(* IEC 61131-3 sources: rusty/examples, 13 files *)

(* ---- pointer.st ---- *)
TYPE MyStruct: STRUCT  x: DINT; y: DINT; END_STRUCT END_TYPE

FUNCTION main : DINT
	main := foo();
END_FUNCTION

FUNCTION foo : DINT
VAR
				x : DINT;
				s : MyStruct;
				u,y : REF_TO DINT;
				z : REF_TO REF_TO DINT;

END_VAR
u := NULL;
u := &s.x;
y := u;
z := &y;
s.x := 9;
z^^ := y^*2;
y^ := z^^*2;

foo := y^;
END_FUNCTION

(* ---- ExternalFunctions.st ---- *)
@EXTERNAL FUNCTION MYLOG : DINT
VAR_INPUT
    x : DINT;
END_VAR
END_FUNCTION

@EXTERNAL FUNCTION MYPRINTF : DINT
VAR_INPUT
    text : STRING;
    value : DINT;
END_VAR
END_FUNCTION

FUNCTION main : DINT
	main := MYLOG(100);
  MYPRINTF('Log value %d\n', main);
END_FUNCTION

(* ---- function_with_return.st ---- *)
FUNCTION smaller_than_ten: BOOL
	VAR_INPUT
		n : INT;
	END_VAR

	IF n < 10 THEN
		smaller_than_ten := TRUE;
		RETURN;
	END_IF;
	smaller_than_ten := FALSE;
END_FUNCTION

(* ---- hello_world.st ---- *)
{external}
FUNCTION puts : DINT
VAR_INPUT {ref}
    text : STRING;
END_VAR
END_FUNCTION

FUNCTION main : DINT
	puts('hello, world!$N');
END_FUNCTION

(* ---- while_loop_with_continue.st ---- *)
FUNCTION main : DINT
  main := 1;
  WHILE main < 10 DO
    main := main + 1;
    CONTINUE;
    main := 200;
  END_WHILE
END_FUNCTION

(* ---- class_method.st ---- *)
CLASS MyClass
    VAR
        x, y : INT;
    END_VAR

    METHOD testMethod
        VAR_INPUT myMethodArg : INT; END_VAR
        VAR myMethodLocalVar : INT; END_VAR

        x := myMethodArg;
    END_METHOD
END_CLASS

(* ---- actions.st ---- *)
PROGRAM main
VAR
	a,b : DINT;
END_VAr

action1();
action2();

END_PROGRAM

ACTIONS
	ACTION action1
		a := a + 1;
	END_ACTION
	ACTION action2
		b := b + 2;
	END_ACTION
END_ACTIONS

(* ---- lt.st ---- *)
FUNCTION a : DINT END_FUNCTION
        PROGRAM main
        VAR
            x : ARRAY[0..1] OF INT;
            y : REF_TO INT;
            z : REF_TO ARRAY[0..1] OF INT;
        END_VAR
            x[0] := 1;
            y^ := 2;
            y^.1 := 3;
            z^[0] := 4;
            z^[1].1 := 5;
						a() := 5;
        END_PROGRAM

(* ---- program_with_expressions.st ---- *)
PROGRAM name
(1 + 2) * (3 + 4);
END_PROGRAM

(* ---- program_with_references.st ---- *)
PROGRAM exp a AND NOT b OR c XOR d; END_PROGRAM

(* ---- program_with_variable_and_operation.st ---- *)
PROGRAM hello
VAR
   x : INT;
   y : INT;
   z : INT;
END_VAR

IF Condition THEN

ELSIF

END_IF;

1 + 2 + 3 + 4;
END_PROGRAM

(* ---- program_with_variables.st ---- *)
PROGRAM hello
VAR
   x : INT
   y : BOOL;
END_VAR
   IF x = 2 THEN
      x := 3
END_PROGRAM

(* ---- simple_program.st ---- *)
PROGRAM prg
    VAR
			a : INT;
			b : REAL;
    END_VAR
		b := 1.5;
		a := b;
END_PROGRAM
